// Mitsubishi GX Works2 project: 2023-04-27 #1   PLC: Q03UDV
// 생산자동화기능사

// global labels: Global1
VAR_GLOBAL
  PB1 AT X0 : BOOL;
  PB2 AT X1 : BOOL;
  정지 AT X2 : BOOL;
  공급후진 AT X3 : BOOL;
  공급전진 AT X4 : BOOL;
  가공후진 AT X5 : BOOL;
  가공전진 AT X6 : BOOL;
  송출후진 AT X7 : BOOL;
  송출전진 AT X8 : BOOL;
  배출후진 AT X9 : BOOL;
  배출전진 AT X0A : BOOL;
  매거진 AT X0B : BOOL;
  금속센서 AT X0F : BOOL;
  PB3 AT X0D : BOOL;
  적색 AT Y20 : BOOL;
  황색 AT Y21 : BOOL;
  녹색 AT Y22 : BOOL;
  공급1 AT Y23 : BOOL;
  공급2 AT Y24 : BOOL;
  가공 AT Y25 : BOOL;
  드릴 AT Y26 : BOOL;
  송출 AT Y27 : BOOL;
  배출 AT Y28 : BOOL;
  컨베이어 AT Y29 : BOOL;
END_VAR

PROGRAM 기본동작
VAR
  STATE : INT;
END_VAR
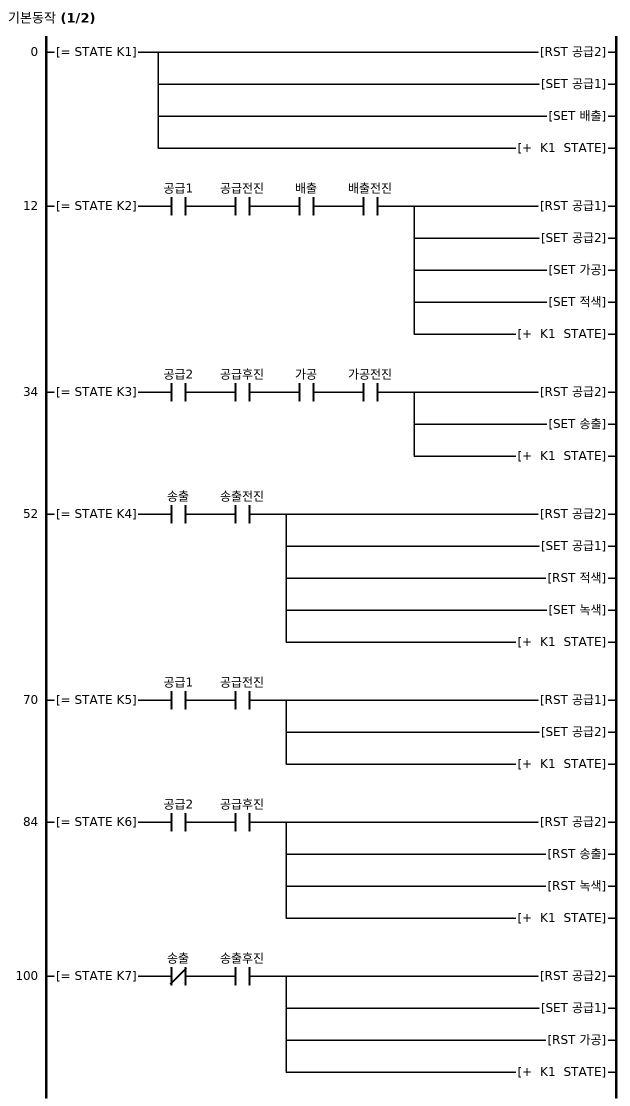
0     LD=     STATE K1
      RST     공급2
      SET     공급1
      SET     배출
      +       K1 STATE
12    LD=     STATE K2
      AND     공급1
      AND     공급전진
      AND     배출
      AND     배출전진
      RST     공급1
      SET     공급2
      SET     가공
      SET     적색
      +       K1 STATE
34    LD=     STATE K3
      AND     공급2
      AND     공급후진
      AND     가공
      AND     가공전진
      RST     공급2
      SET     송출
      +       K1 STATE
52    LD=     STATE K4
      AND     송출
      AND     송출전진
      RST     공급2
      SET     공급1
      RST     적색
      SET     녹색
      +       K1 STATE
70    LD=     STATE K5
      AND     공급1
      AND     공급전진
      RST     공급1
      SET     공급2
      +       K1 STATE
84    LD=     STATE K6
      AND     공급2
      AND     공급후진
      RST     공급2
      RST     송출
      RST     녹색
      +       K1 STATE
100   LD=     STATE K7
      ANI     송출
      AND     송출후진
      RST     공급2
      SET     공급1
      RST     가공
      +       K1 STATE
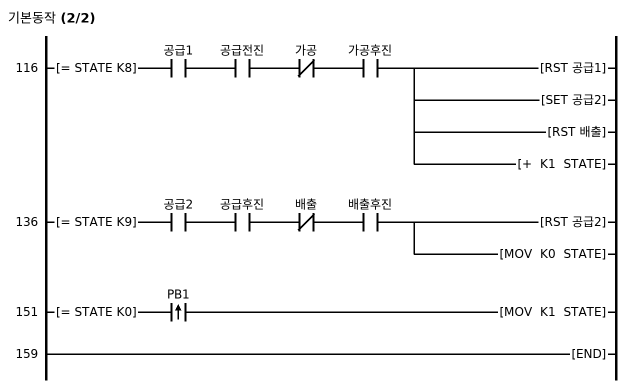
116   LD=     STATE K8
      AND     공급1
      AND     공급전진
      ANI     가공
      AND     가공후진
      RST     공급1
      SET     공급2
      RST     배출
      +       K1 STATE
136   LD=     STATE K9
      AND     공급2
      AND     공급후진
      ANI     배출
      AND     배출후진
      RST     공급2
      MOV     K0 STATE
151   LD=     STATE K0
      ANDP    PB1
      MOV     K1 STATE
159   END
END_PROGRAM

PROGRAM 응용동작1
VAR
  STATE : INT;
END_VAR
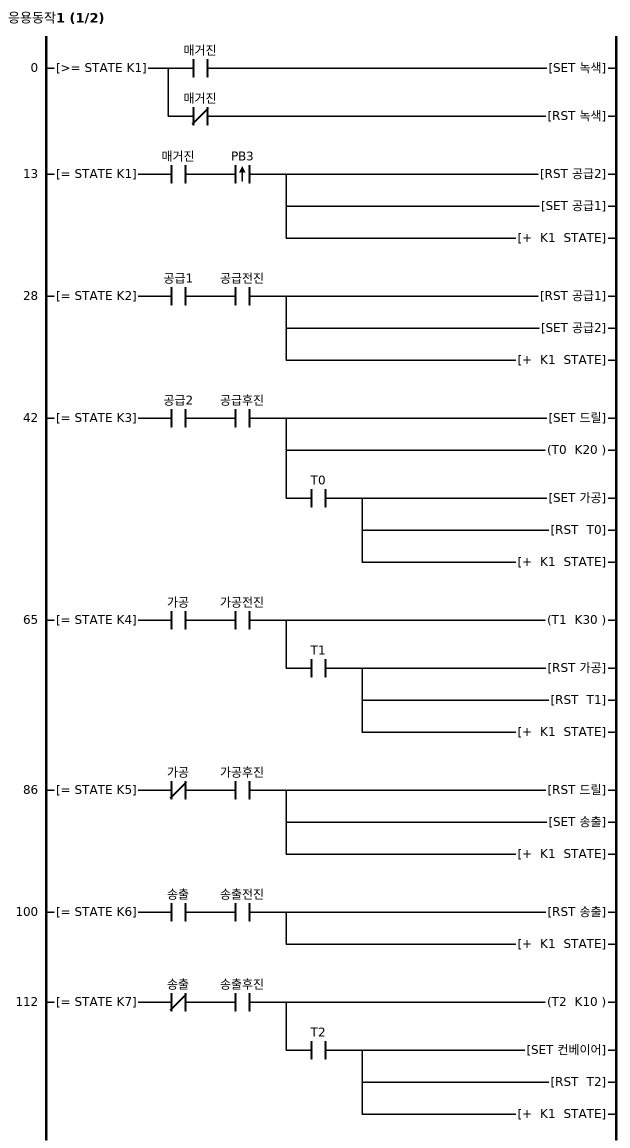
0     LD>=    STATE K1
      MPS
      AND     매거진
      SET     녹색
      MPP
      ANI     매거진
      RST     녹색
13    LD=     STATE K1
      AND     매거진
      ANDP    PB3
      RST     공급2
      SET     공급1
      +       K1 STATE
28    LD=     STATE K2
      AND     공급1
      AND     공급전진
      RST     공급1
      SET     공급2
      +       K1 STATE
42    LD=     STATE K3
      AND     공급2
      AND     공급후진
      SET     드릴
      OUT     T0 K20
      AND     T0
      SET     가공
      RST     T0
      +       K1 STATE
65    LD=     STATE K4
      AND     가공
      AND     가공전진
      OUT     T1 K30
      AND     T1
      RST     가공
      RST     T1
      +       K1 STATE
86    LD=     STATE K5
      ANI     가공
      AND     가공후진
      RST     드릴
      SET     송출
      +       K1 STATE
100   LD=     STATE K6
      AND     송출
      AND     송출전진
      RST     송출
      +       K1 STATE
112   LD=     STATE K7
      ANI     송출
      AND     송출후진
      OUT     T2 K10
      AND     T2
      SET     컨베이어
      RST     T2
      +       K1 STATE
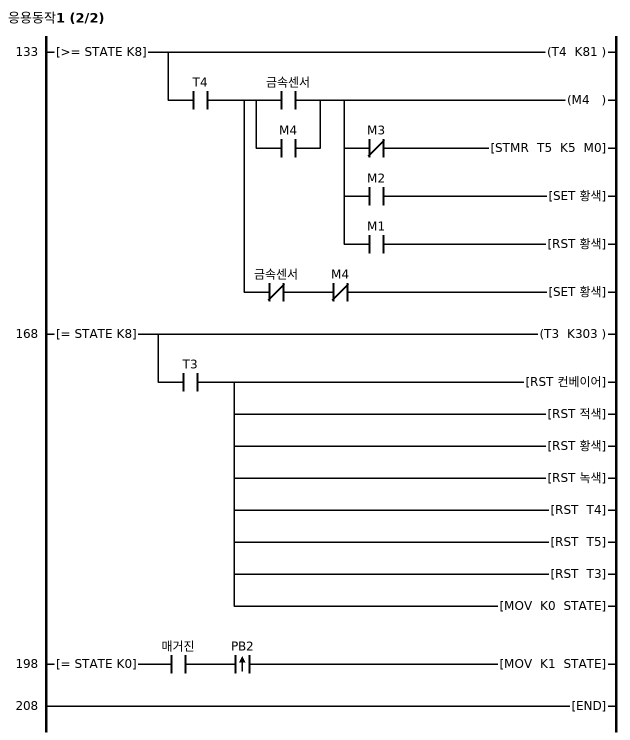
133   LD>=    STATE K8
      OUT     T4 K81
      AND     T4
      MPS
      LD      금속센서
      OR      M4
      ANB
      OUT     M4
      MPS
      ANI     M3
      STMR    T5 K5 M0
      MRD
      AND     M2
      SET     황색
      MPP
      AND     M1
      RST     황색
      MPP
      ANI     금속센서
      ANI     M4
      SET     황색
168   LD=     STATE K8
      OUT     T3 K303
      AND     T3
      RST     컨베이어
      RST     적색
      RST     황색
      RST     녹색
      RST     T4
      RST     T5
      RST     T3
      MOV     K0 STATE
198   LD=     STATE K0
      AND     매거진
      ANDP    PB2
      MOV     K1 STATE
208   END
END_PROGRAM

PROGRAM 응용동작2
VAR
  STATE : INT;
END_VAR
0     END
END_PROGRAM
